TYPE T_Generic : __SYSTEM.AnyType ; END_TYPE

(* stored: Version 1.1.0.1
   DUT T_Generic: Id {13d55dd5-dc13-4a22-b434-03436eac97d3} *)
